INTERFACE I_InterfaceDatatype_ITcVnImage EXTENDS I_InterfaceDatatype

PROPERTY PUBLIC Value : REFERENCE TO ITcVnImage
GET
END_GET
END_PROPERTY

END_INTERFACE

(* stored: Version 1.1.0.1, ProductVersion 3.1.4024.13
   Itf I_InterfaceDatatype_ITcVnImage: Id {32424d8f-1289-06d5-2086-127d40c72a01}
   Property Value: Id {26c8a13c-cffd-0ff2-190b-2bd6b2cb977f}
   Get Get: Id {66022c92-aabf-0cfc-2510-659901115904} *)
